// Mitsubishi GX Works2 project: modbus slave- training   PLC: FX3U/FX3UC

PROGRAM MAIN
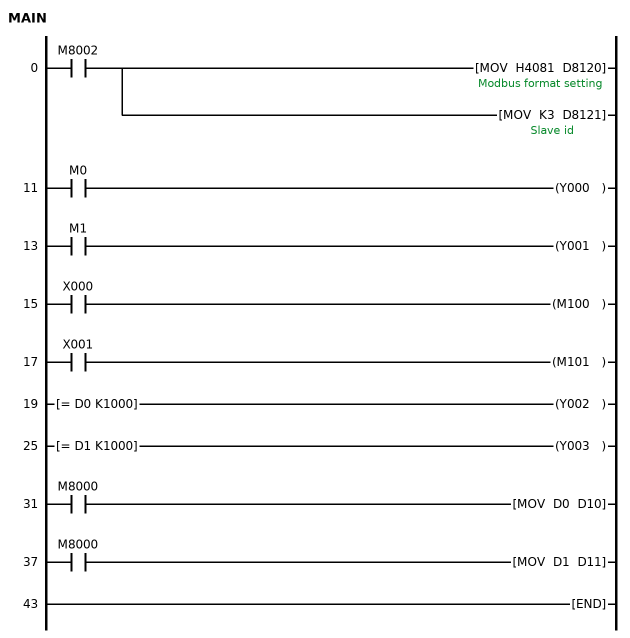
0     LD      M8002
      MOV     H4081 D8120  ; Modbus format setting
      MOV     K3 D8121  ; Slave id
11    LD      M0
      OUT     Y000
13    LD      M1
      OUT     Y001
15    LD      X000
      OUT     M100
17    LD      X001
      OUT     M101
19    LD=     D0 K1000
      OUT     Y002
25    LD=     D1 K1000
      OUT     Y003
31    LD      M8000
      MOV     D0 D10
37    LD      M8000
      MOV     D1 D11
43    END
END_PROGRAM
